(* PLC project Untitled6.project, CODESYS CODESYS V3.5 SP20 *)
(* stored: creationDateTime 2025-11-22T16:58:05.889821, modificationDateTime 2025-11-22T16:57:51.3762535 *)

TYPE ST_MotionState : STRUCT
  fDuration : LREAL := 0.0;  (* Duration of this segment *)
  fPos : LREAL := 0.0;  (* Position *)
  fVel : LREAL := 0.0;  (* Velocity *)
  fAcc : LREAL := 0.0;  (* Acceleration *)
  fJerk : LREAL := 0.0;  (* Jerk *)
END_STRUCT;
END_TYPE

TYPE ST_MotionLimits : STRUCT
  fVelMax : LREAL;
  fAccMax : LREAL;
  fJerkMax : LREAL;
END_STRUCT;
END_TYPE

FUNCTION FC_S7RTT_CalcTrajDist : LREAL
  VAR_INPUT
    v_peak : LREAL;
    start_v : LREAL;
    start_a : LREAL;
    target_v : LREAL;
    a_max : LREAL;
    j_max : LREAL;
  END_VAR
  VAR
    t_buf : ARRAY[1..5] OF LREAL;
    j_buf : ARRAY[1..5] OF LREAL;
    cnt : INT;
    i : INT;
    v_curr : LREAL;
    a_curr : LREAL;
    dist_total : LREAL;
    t_seg : LREAL;
    j_seg : LREAL;
  END_VAR

            dist_total := 0.0;
v_curr := start_v;
a_curr := start_a;

// Phase 1: Start -> Peak Velocity
cnt := FC_S7RTT_BuildProfile(v_curr, a_curr, v_peak, a_max, j_max, t_buf, j_buf);
FOR i := 1 TO cnt DO
	t_seg := t_buf[i];
	j_seg := j_buf[i];
    // Standard kinematic integration: p = p0 + v0*t + 0.5*a0*t^2 + 1/6*j*t^3
	dist_total := dist_total + v_curr * t_seg + 0.5 * a_curr * t_seg*t_seg + (1.0/6.0) * j_seg * t_seg*t_seg*t_seg;
	v_curr := v_curr + a_curr * t_seg + 0.5 * j_seg * t_seg*t_seg;
	a_curr := a_curr + j_seg * t_seg;
END_FOR;

// Phase 2: Peak Velocity -> Target Velocity
cnt := FC_S7RTT_BuildProfile(v_curr, a_curr, target_v, a_max, j_max, t_buf, j_buf);
FOR i := 1 TO cnt DO
	t_seg := t_buf[i];
	j_seg := j_buf[i];
	dist_total := dist_total + v_curr * t_seg + 0.5 * a_curr * t_seg*t_seg + (1.0/6.0) * j_seg * t_seg*t_seg*t_seg;
	v_curr := v_curr + a_curr * t_seg + 0.5 * j_seg * t_seg*t_seg;
	a_curr := a_curr + j_seg * t_seg;
END_FOR;

FC_S7RTT_CalcTrajDist := dist_total;
          
END_FUNCTION

FUNCTION_BLOCK FB_S7RTT_Plan
  VAR_INPUT
    Execute : BOOL;
    ModeVelocity : BOOL;
    StartState : ST_MotionState;
    TargetPos : LREAL;
    TargetVel : LREAL;
    Limits : ST_MotionLimits;
  END_VAR
  VAR_OUTPUT
    Done : BOOL;
    Error : BOOL;
    SegmentCount : INT;
    Trajectory : ARRAY[1..32] OF ST_MotionState;
  END_VAR
  VAR
    trig_exec : BOOL;
    prev_exec : BOOL;
    c_pos : LREAL;
    c_vel : LREAL;
    c_acc : LREAL;
    dist_req : LREAL;
    iter : INT;
    sa : LREAL;
    sb : LREAL;
    sc : LREAL;
    fa : LREAL;
    fb : LREAL;
    fc : LREAL;
    sd : LREAL;
    se : LREAL;
    tol1 : LREAL;
    xm : LREAL;
    fCoefP : LREAL;
    fCoefQ : LREAL;
    fCoefR : LREAL;
    fCoefS : LREAL;
    min1 : LREAL;
    min2 : LREAL;
    mflag : BOOL;
    best_v : LREAL;
    t_shape_buf : ARRAY[1..5] OF LREAL;
    j_shape_buf : ARRAY[1..5] OF LREAL;
    shape_cnt : INT;
    i : INT;
    t_rec : LREAL;
    d_upper : LREAL;
    d_lower : LREAL;
    d_inertial : LREAL;
    v_inertial : LREAL;
    j_restore : LREAL;
    t_to_zero : LREAL;
    gap : LREAL;
    t_cruise : LREAL;
    v_mid : LREAL;
    a_mid : LREAL;
    EPS_TIME : LREAL := 1E-09;
    EPS_VAL : LREAL := 1E-07;
    EPS_ACC : LREAL := 1E-06;
    EPS_DIST : LREAL := 1E-08;
    SOLVER_TOL : LREAL := 1E-08;
    SOLVER_EPS : LREAL := 2.22E-16;
    MAX_ITER : INT := 100;
    ref_idx : INT;
    max_dt : LREAL;
    dt_fix : LREAL;
    v_cruise_start : LREAL;
    new_dt : LREAL;
  END_VAR

            // ==============================================================================
// File Name:    FB_S7RTT_Plan.st
// Author:       feecat
// Version:      V1.6.1
// Description:  Simple 7seg Real-Time Trajectory Generator
// Website:      https://github.com/feecat/S7RTT
// License:      Apache License Version 2.0
// ==============================================================================
//
// Licensed under the Apache License, Version 2.0 (the "License");
// you may not use this file except in compliance with the License.
// You may obtain a copy of the License at
//
//     http://www.apache.org/licenses/LICENSE-2.0
//
// Unless required by applicable law or agreed to in writing, software
// distributed under the License is distributed on an "AS IS" BASIS,
// WITHOUT WARRANTIES OR CONDITIONS OF ANY KIND, either express or implied.
// See the License for the specific language governing permissions and
// limitations under the License.
// ==============================================================================

trig_exec := Execute AND NOT prev_exec;
prev_exec := Execute;

IF NOT Execute THEN
	Done := FALSE;
	Error := FALSE;
	RETURN;
END_IF

IF NOT trig_exec THEN
	RETURN;
END_IF;

// --- Initialization ---
Done := FALSE;
Error := FALSE;
SegmentCount := 0;

IF Limits.fVelMax <= 0.0 OR Limits.fAccMax <= 0.0 OR Limits.fJerkMax <= 0.0 THEN
	Error := TRUE;
	RETURN;
END_IF;

c_pos := StartState.fPos;
c_vel := StartState.fVel;
c_acc := StartState.fAcc;

// ========================================================
// 1. Acceleration Recovery (Safety Decel to Max Limits)
// ========================================================
IF c_acc > Limits.fAccMax + EPS_VAL THEN
	t_rec := (c_acc - Limits.fAccMax) / Limits.fJerkMax;
	SegmentCount := SegmentCount + 1;
	Trajectory[SegmentCount].fDuration := t_rec;
	Trajectory[SegmentCount].fJerk     := -Limits.fJerkMax;
	
	// Integrate state forward
	c_pos := c_pos + c_vel * t_rec + 0.5 * c_acc * t_rec*t_rec + (1.0/6.0) * (-Limits.fJerkMax) * t_rec*t_rec*t_rec;
	c_vel := c_vel + c_acc * t_rec + 0.5 * (-Limits.fJerkMax) * t_rec*t_rec;
	c_acc := Limits.fAccMax;
	
ELSIF c_acc < -Limits.fAccMax - EPS_VAL THEN
	t_rec := (-Limits.fAccMax - c_acc) / Limits.fJerkMax;
	SegmentCount := SegmentCount + 1;
	Trajectory[SegmentCount].fDuration := t_rec;
	Trajectory[SegmentCount].fJerk     := Limits.fJerkMax;
	
	// Integrate state forward
	c_pos := c_pos + c_vel * t_rec + 0.5 * c_acc * t_rec*t_rec + (1.0/6.0) * (Limits.fJerkMax) * t_rec*t_rec*t_rec;
	c_vel := c_vel + c_acc * t_rec + 0.5 * (Limits.fJerkMax) * t_rec*t_rec;
	c_acc := -Limits.fAccMax;
END_IF;

// ========================================================
// 2. Plan Generation
// ========================================================

IF ModeVelocity THEN
	// ---------------- Velocity Mode ----------------
	v_mid := TargetVel; 
	IF v_mid > Limits.fVelMax THEN v_mid := Limits.fVelMax; END_IF;
	IF v_mid < -Limits.fVelMax THEN v_mid := -Limits.fVelMax; END_IF;

	shape_cnt := FC_S7RTT_BuildProfile(c_vel, c_acc, v_mid, Limits.fAccMax, Limits.fJerkMax, t_shape_buf, j_shape_buf);
	
	FOR i := 1 TO shape_cnt DO
		IF SegmentCount < 32 THEN
			SegmentCount := SegmentCount + 1;
			Trajectory[SegmentCount].fDuration := t_shape_buf[i];
			Trajectory[SegmentCount].fJerk     := j_shape_buf[i];
		END_IF;
	END_FOR;

ELSE
	// ---------------- Position Mode ----------------
	dist_req := TargetPos - c_pos;
	
	// Calculate Inertial Velocity (Peak velocity if we stopped now)
	t_to_zero := ABS(c_acc) / Limits.fJerkMax;
	IF c_acc > 0.0 THEN j_restore := -Limits.fJerkMax; ELSE j_restore := Limits.fJerkMax; END_IF;
	v_inertial := c_vel + c_acc * t_to_zero + 0.5 * j_restore * t_to_zero * t_to_zero;

	// Check 1: Max Reach Checks (Can we physically reach the target?)
	// This determines if we need to cruise at VMax
	d_upper := FC_S7RTT_CalcTrajDist(Limits.fVelMax, c_vel, c_acc, TargetVel, Limits.fAccMax, Limits.fJerkMax);
	d_lower := FC_S7RTT_CalcTrajDist(-Limits.fVelMax, c_vel, c_acc, TargetVel, Limits.fAccMax, Limits.fJerkMax);

	IF dist_req > d_upper + EPS_DIST THEN
		// Case: Cruise Positive (Go to Vmax, Cruise, then Decel)
		gap := dist_req - d_upper;
		t_cruise := gap / Limits.fVelMax;
		
		// 1. Start -> Vmax
		shape_cnt := FC_S7RTT_BuildProfile(c_vel, c_acc, Limits.fVelMax, Limits.fAccMax, Limits.fJerkMax, t_shape_buf, j_shape_buf);
		
		// Add Cruise Segment
		IF t_cruise > EPS_TIME THEN
		   shape_cnt := shape_cnt + 1;
		   t_shape_buf[shape_cnt] := t_cruise;
		   j_shape_buf[shape_cnt] := 0.0;
		END_IF;
		
		// Integ & Append
		v_mid := c_vel; a_mid := c_acc;
		FOR i := 1 TO shape_cnt DO
			IF SegmentCount < 32 THEN
				SegmentCount := SegmentCount + 1;
				Trajectory[SegmentCount].fDuration := t_shape_buf[i];
				Trajectory[SegmentCount].fJerk     := j_shape_buf[i];
				v_mid := v_mid + a_mid * t_shape_buf[i] + 0.5 * j_shape_buf[i] * t_shape_buf[i]*t_shape_buf[i];
				a_mid := a_mid + j_shape_buf[i] * t_shape_buf[i];
			END_IF;
		END_FOR;
		
		// 2. Vmax -> Target
		shape_cnt := FC_S7RTT_BuildProfile(v_mid, a_mid, TargetVel, Limits.fAccMax, Limits.fJerkMax, t_shape_buf, j_shape_buf);
		FOR i := 1 TO shape_cnt DO
			IF SegmentCount < 32 THEN
				SegmentCount := SegmentCount + 1;
				Trajectory[SegmentCount].fDuration := t_shape_buf[i];
				Trajectory[SegmentCount].fJerk     := j_shape_buf[i];
			END_IF;
		END_FOR;

	ELSIF dist_req < d_lower - EPS_DIST THEN
		// Case: Cruise Negative
		gap := dist_req - d_lower;
		t_cruise := gap / (-Limits.fVelMax);
		
		// 1. Start -> -Vmax
		shape_cnt := FC_S7RTT_BuildProfile(c_vel, c_acc, -Limits.fVelMax, Limits.fAccMax, Limits.fJerkMax, t_shape_buf, j_shape_buf);
		
		IF t_cruise > EPS_TIME THEN
		   shape_cnt := shape_cnt + 1;
		   t_shape_buf[shape_cnt] := t_cruise;
		   j_shape_buf[shape_cnt] := 0.0;
		END_IF;
		
		v_mid := c_vel; a_mid := c_acc;
		FOR i := 1 TO shape_cnt DO
			IF SegmentCount < 32 THEN
				SegmentCount := SegmentCount + 1;
				Trajectory[SegmentCount].fDuration := t_shape_buf[i];
				Trajectory[SegmentCount].fJerk     := j_shape_buf[i];
				v_mid := v_mid + a_mid * t_shape_buf[i] + 0.5 * j_shape_buf[i] * t_shape_buf[i]*t_shape_buf[i];
				a_mid := a_mid + j_shape_buf[i] * t_shape_buf[i];
			END_IF;
		END_FOR;
		
		// 2. -Vmax -> Target
		shape_cnt := FC_S7RTT_BuildProfile(v_mid, a_mid, TargetVel, Limits.fAccMax, Limits.fJerkMax, t_shape_buf, j_shape_buf);
		FOR i := 1 TO shape_cnt DO
			IF SegmentCount < 32 THEN
				SegmentCount := SegmentCount + 1;
				Trajectory[SegmentCount].fDuration := t_shape_buf[i];
				Trajectory[SegmentCount].fJerk     := j_shape_buf[i];
			END_IF;
		END_FOR;

	ELSE
		// Case: Target is reachable without cruising at limits. 
		// We need to find the peak velocity 'v_peak' that produces the exact distance.
		
		d_inertial := FC_S7RTT_CalcTrajDist(v_inertial, c_vel, c_acc, TargetVel, Limits.fAccMax, Limits.fJerkMax);
		
		// Define search brackets for Brent's method [sa, sb]
		// Logic: If requested distance > inertial distance, we need to go faster/more positive.
		IF dist_req > d_inertial THEN
			sa := v_inertial - (10.0 * EPS_VAL);
			sb := MAX(Limits.fVelMax, MAX(ABS(c_vel), ABS(TargetVel))) * 1.5 + 10.0;
		ELSE
			sb := v_inertial + (10.0 * EPS_VAL);
			sa := -(MAX(Limits.fVelMax, MAX(ABS(c_vel), ABS(TargetVel))) * 1.5 + 10.0);
		END_IF;
		
		IF sa >= sb THEN sa := sb - EPS_VAL; END_IF;
		
		// Function evaluation at endpoints
		fa := FC_S7RTT_CalcTrajDist(sa, c_vel, c_acc, TargetVel, Limits.fAccMax, Limits.fJerkMax) - dist_req;
		fb := FC_S7RTT_CalcTrajDist(sb, c_vel, c_acc, TargetVel, Limits.fAccMax, Limits.fJerkMax) - dist_req;
		
		IF (fa > 0.0 AND fb > 0.0) OR (fa < 0.0 AND fb < 0.0) THEN
			// Error: Root not bracketed. Use the best guess.
			IF ABS(fa) < ABS(fb) THEN best_v := sa; ELSE best_v := sb; END_IF;
		ELSE
			// Brent's Method Solver
			sc := sa; fc := fa; sd := sb - sa; se := sd; mflag := TRUE;
			
			FOR iter := 1 TO MAX_ITER DO
				 IF ABS(fc) < ABS(fb) THEN
					sa := sb; sb := sc; sc := sa;
					fa := fb; fb := fc; fc := fa;
				 END_IF;
				 
				 tol1 := 2.0 * SOLVER_EPS * ABS(sb) + 0.5 * SOLVER_TOL;
				 xm := 0.5 * (sc - sb);
				 
				 IF ABS(xm) <= tol1 OR ABS(fb) < SOLVER_TOL THEN
					EXIT; // Converged
				 END_IF;
				 
				 IF ABS(se) >= tol1 AND ABS(fa) > ABS(fb) THEN
					fCoefS := fb / fa;
					IF sa = sc THEN
						fCoefP := 2.0 * xm * fCoefS;
						fCoefQ := 1.0 - fCoefS;
					ELSE
						fCoefQ := fa / fc; fCoefR := fb / fc;
						fCoefP := fCoefS * (2.0 * xm * fCoefQ * (fCoefQ - fCoefR) - (sb - sa) * (fCoefR - 1.0));
						fCoefQ := (fCoefQ - 1.0) * (fCoefR - 1.0) * (fCoefS - 1.0);
					END_IF;
					
					IF fCoefP > 0.0 THEN fCoefQ := -fCoefQ; END_IF;
					fCoefP := ABS(fCoefP);
					min1 := 3.0 * xm * fCoefQ - ABS(tol1 * fCoefQ);
					min2 := ABS(se * fCoefQ);
					
					IF 2.0 * fCoefP < min1 THEN
						IF mflag THEN
							IF 2.0 * fCoefP < min2 THEN se := sd; sd := fCoefP / fCoefQ; mflag := FALSE;
							ELSE sd := xm; se := sd; mflag := TRUE; END_IF;
						ELSE
							IF 2.0 * fCoefP < ABS(sd * fCoefQ) THEN se := sd; sd := fCoefP / fCoefQ; mflag := FALSE;
							ELSE sd := xm; se := sd; mflag := TRUE; END_IF;
						END_IF;
					ELSE
						sd := xm; se := sd; mflag := TRUE;
					END_IF;
				 ELSE
					 sd := xm; se := sd; mflag := TRUE;
				 END_IF;
				 
				 sa := sb; fa := fb;
				 
				 IF ABS(sd) > tol1 THEN
					sb := sb + sd;
				 ELSE
					IF xm > 0.0 THEN sb := sb + tol1; ELSE sb := sb - tol1; END_IF;
				 END_IF;
				 
				 fb := FC_S7RTT_CalcTrajDist(sb, c_vel, c_acc, TargetVel, Limits.fAccMax, Limits.fJerkMax) - dist_req;
				 
				 IF (fb > 0.0 AND fc > 0.0) OR (fb < 0.0 AND fc < 0.0) THEN
					 sc := sa; fc := fa; sd := sb - sa; se := sd; mflag := TRUE;
				 END_IF;
			END_FOR;
			best_v := sb;
		END_IF;
		
		// Generate final trajectory using the solved velocity
		// 1. Start -> v_peak
		shape_cnt := FC_S7RTT_BuildProfile(c_vel, c_acc, best_v, Limits.fAccMax, Limits.fJerkMax, t_shape_buf, j_shape_buf);
		v_mid := c_vel; a_mid := c_acc;
		FOR i := 1 TO shape_cnt DO
			IF SegmentCount < 32 THEN
				SegmentCount := SegmentCount + 1;
				Trajectory[SegmentCount].fDuration := t_shape_buf[i];
				Trajectory[SegmentCount].fJerk     := j_shape_buf[i];
				v_mid := v_mid + a_mid * t_shape_buf[i] + 0.5 * j_shape_buf[i] * t_shape_buf[i]*t_shape_buf[i];
				a_mid := a_mid + j_shape_buf[i] * t_shape_buf[i];
			END_IF;
		END_FOR;
		
		// 2. v_peak -> Target
		shape_cnt := FC_S7RTT_BuildProfile(v_mid, a_mid, TargetVel, Limits.fAccMax, Limits.fJerkMax, t_shape_buf, j_shape_buf);
		FOR i := 1 TO shape_cnt DO
			IF SegmentCount < 32 THEN
				SegmentCount := SegmentCount + 1;
				Trajectory[SegmentCount].fDuration := t_shape_buf[i];
				Trajectory[SegmentCount].fJerk     := j_shape_buf[i];
			END_IF;
		END_FOR;
	END_IF; // End Bounds Checks
END_IF; // End ModeVelocity
// ========================================================
// 2.5. Trajectory Refinement (Fix Integration Drift)
// ========================================================
// Only perform refinement if we have segments and are in Position Mode
IF SegmentCount > 0 AND NOT ModeVelocity THEN
	c_pos := StartState.fPos;
	c_vel := StartState.fVel;
	c_acc := StartState.fAcc;
	
	// Variables for refinement search
	// You need to declare: 
	// ref_idx: INT; max_dt: LREAL; sim_p: LREAL; 
	// dt_fix: LREAL; v_cruise_start: LREAL;
	
	ref_idx := -1;
	max_dt := -1.0;
	
	FOR i := 1 TO SegmentCount DO
		t_rec := Trajectory[i].fDuration;
		j_restore := Trajectory[i].fJerk;
		
		// Check for Constant Velocity segment (J=0, A approx 0)
		// We simulate A at the START of the segment
		IF ABS(j_restore) < SOLVER_EPS AND ABS(c_acc) < EPS_ACC THEN
			IF t_rec > max_dt THEN
				max_dt := t_rec;
				ref_idx := i;
				v_cruise_start := c_vel; // Store velocity of this segment
			END_IF;
		END_IF;
		
		// Integrate to next state
		c_pos := c_pos + c_vel * t_rec + 0.5 * c_acc * t_rec*t_rec + (1.0/6.0) * j_restore * t_rec*t_rec*t_rec;
		c_vel := c_vel + c_acc * t_rec + 0.5 * j_restore * t_rec*t_rec;
		c_acc := c_acc + j_restore * t_rec;
	END_FOR;
	
	// Calculate Error based on simulated final position
	gap := TargetPos - c_pos;
	
	// Apply fix if we found a suitable cruise segment and error exists
	IF ref_idx <> -1 AND ABS(gap) > EPS_DIST AND ABS(v_cruise_start) > EPS_VAL THEN
		dt_fix := gap / v_cruise_start;
		Trajectory[ref_idx].fDuration := Trajectory[ref_idx].fDuration + dt_fix;
		
		// Safety: prevent negative time
		IF Trajectory[ref_idx].fDuration < EPS_TIME THEN 
			Trajectory[ref_idx].fDuration := EPS_TIME; 
		END_IF;
	END_IF;
END_IF;

// ========================================================
// 3. Final Pass: Calculate Absolute Positions
// ========================================================
c_pos := StartState.fPos; 
c_vel := StartState.fVel; 
c_acc := StartState.fAcc;

FOR i := 1 TO SegmentCount DO
	// Store the starting state of this segment
	Trajectory[i].fPos := c_pos;
	Trajectory[i].fVel := c_vel;
	Trajectory[i].fAcc := c_acc;
	
	t_rec := Trajectory[i].fDuration;
	j_restore := Trajectory[i].fJerk;
	
	c_pos := c_pos + c_vel * t_rec + 0.5 * c_acc * t_rec*t_rec + (1.0/6.0) * j_restore * t_rec*t_rec*t_rec;
	c_vel := c_vel + c_acc * t_rec + 0.5 * j_restore * t_rec*t_rec;
	c_acc := c_acc + j_restore * t_rec;
END_FOR;

Done := TRUE;
          
END_FUNCTION_BLOCK

FUNCTION FC_S7RTT_AtTime : ST_MotionState
  VAR_INPUT
    Trajectory : ARRAY[1..32] OF ST_MotionState;
    SegCount : INT;
    ElapsedTime : LREAL;
  END_VAR
  VAR
    i : INT;
    t_rem : LREAL;
    t : LREAL;
    j : LREAL;
    p0 : LREAL;
    v0 : LREAL;
    a0 : LREAL;
    last_idx : INT;
  END_VAR

            IF SegCount <= 0 THEN
    // No trajectory, return zero/empty state
    FC_S7RTT_AtTime.fPos := 0.0; FC_S7RTT_AtTime.fVel := 0.0; FC_S7RTT_AtTime.fAcc := 0.0;
    RETURN;
END_IF;

IF ElapsedTime <= 0.0 THEN
     // Return Initial State from First Segment
     FC_S7RTT_AtTime := Trajectory[1]; 
     FC_S7RTT_AtTime.fDuration := 0.0;
     FC_S7RTT_AtTime.fJerk := 0.0;
     RETURN;
END_IF;

t_rem := ElapsedTime;

FOR i := 1 TO SegCount DO
	IF t_rem <= Trajectory[i].fDuration THEN
		t := t_rem;
		j := Trajectory[i].fJerk;
		// Use pre-calculated state at segment start
		p0 := Trajectory[i].fPos;
		v0 := Trajectory[i].fVel;
		a0 := Trajectory[i].fAcc;

		FC_S7RTT_AtTime.fPos := p0 + v0 * t + 0.5 * a0 * t*t + (1.0/6.0) * j * t*t*t;
		FC_S7RTT_AtTime.fVel := v0 + a0 * t + 0.5 * j * t*t;
		FC_S7RTT_AtTime.fAcc := a0 + j * t;
		FC_S7RTT_AtTime.fJerk := j;
		FC_S7RTT_AtTime.fDuration := 0.0;
		RETURN;
	ELSE
		t_rem := t_rem - Trajectory[i].fDuration;
	END_IF;
END_FOR;

// Time is beyond end of trajectory
// Calculate Final State of last segment
last_idx := SegCount;
t := Trajectory[last_idx].fDuration;
j := Trajectory[last_idx].fJerk;
p0 := Trajectory[last_idx].fPos;
v0 := Trajectory[last_idx].fVel;
a0 := Trajectory[last_idx].fAcc;

p0 := p0 + v0 * t + 0.5 * a0 * t*t + (1.0/6.0) * j * t*t*t;
v0 := v0 + a0 * t + 0.5 * j * t*t;

// Hold Final Position (assuming v=target, a=0 at end)
// Linear projection if Velocity is non-zero
FC_S7RTT_AtTime.fPos := p0 + v0 * t_rem;
FC_S7RTT_AtTime.fVel := v0;
FC_S7RTT_AtTime.fAcc := 0.0;
FC_S7RTT_AtTime.fJerk := 0.0;
FC_S7RTT_AtTime.fDuration := 0.0;
          
END_FUNCTION

FUNCTION FC_S7RTT_BuildProfile : INT
  VAR_INPUT
    in_v_start : LREAL;
    in_a_start : LREAL;
    in_v_target : LREAL;
    in_a_max : LREAL;
    in_j_max : LREAL;
  END_VAR
  VAR_IN_OUT
    out_time : ARRAY[1..5] OF LREAL;
    out_jerk : ARRAY[1..5] OF LREAL;
  END_VAR
  VAR
    acc_clamped : LREAL;
    t_to_zero : LREAL;
    j_restore : LREAL;
    v_min_feasible : LREAL;
    direction : LREAL;
    v0_mod : LREAL;
    a0_mod : LREAL;
    v1_mod : LREAL;
    t1_max : LREAL;
    t3_max : LREAL;
    dv_inflection : LREAL;
    dv_req : LREAL;
    dv_missing : LREAL;
    term : LREAL;
    a_peak : LREAL;
    t1 : LREAL;
    t2 : LREAL;
    t3 : LREAL;
    cnt : INT;
    EPS : LREAL := 1E-09;
  END_VAR

            cnt := 0;

// 1. Clamp initial acceleration to limits
acc_clamped := in_a_start;
IF acc_clamped > in_a_max THEN acc_clamped := in_a_max; END_IF;
IF acc_clamped < -in_a_max THEN acc_clamped := -in_a_max; END_IF;

// 2. Check feasibility (can we stop?)
t_to_zero := ABS(acc_clamped) / in_j_max;
IF ABS(acc_clamped) > EPS THEN
    IF acc_clamped > 0.0 THEN j_restore := -in_j_max; ELSE j_restore := in_j_max; END_IF;
ELSE
    j_restore := 0.0;
END_IF;

v_min_feasible := in_v_start + acc_clamped * t_to_zero + 0.5 * j_restore * t_to_zero * t_to_zero;

// 3. Determine direction
direction := 1.0;
IF in_v_target < v_min_feasible - EPS THEN
    direction := -1.0;
END_IF;

// 4. Normalize to positive quadrant
v0_mod := in_v_start * direction;
a0_mod := acc_clamped * direction;
v1_mod := in_v_target * direction;

t1_max := (in_a_max - a0_mod) / in_j_max;
IF t1_max < 0.0 THEN t1_max := 0.0; END_IF;

t3_max := in_a_max / in_j_max;

// Velocity change at inflection (max accel reached)
dv_inflection := (a0_mod * t1_max + 0.5 * in_j_max * t1_max * t1_max) +
                 (in_a_max * t3_max - 0.5 * in_j_max * t3_max * t3_max);

dv_req := v1_mod - v0_mod;

// 5. Calculate profile times
IF dv_req > dv_inflection THEN
    // Trapezoidal (Constant Acceleration Phase)
    dv_missing := dv_req - dv_inflection;
    t2 := dv_missing / in_a_max;
    t1 := t1_max;
    t3 := t3_max;
ELSE
    // Triangular (No Constant Acceleration)
    term := in_j_max * dv_req + 0.5 * a0_mod * a0_mod;
    IF term < 0.0 THEN term := 0.0; END_IF;
    a_peak := SQRT(term);
    
    t1 := (a_peak - a0_mod) / in_j_max;
    IF t1 < 0.0 THEN t1 := 0.0; END_IF;
    
    t3 := a_peak / in_j_max;
    IF t3 < 0.0 THEN t3 := 0.0; END_IF;
    
    t2 := 0.0;
END_IF;

// 6. Output Segments
IF t1 > EPS THEN
    cnt := cnt + 1; out_time[cnt] := t1; out_jerk[cnt] := direction * in_j_max;
END_IF;
IF t2 > EPS THEN
    cnt := cnt + 1; out_time[cnt] := t2; out_jerk[cnt] := 0.0;
END_IF;
IF t3 > EPS THEN
    cnt := cnt + 1; out_time[cnt] := t3; out_jerk[cnt] := -direction * in_j_max;
END_IF;

FC_S7RTT_BuildProfile := cnt;
          
END_FUNCTION

FUNCTION_BLOCK FB_S7RTT_Plan_Velocity
  VAR_INPUT
    Execute : BOOL;
    StartState : ST_MotionState;
    TargetVel : LREAL;
    Limits : ST_MotionLimits;
  END_VAR
  VAR_OUTPUT
    Done : BOOL;
    Error : BOOL;
    SegmentCount : INT;
    Trajectory : ARRAY[1..32] OF ST_MotionState;
  END_VAR
  VAR
    trig_exec : BOOL;
    prev_exec : BOOL;
    c_pos : LREAL;
    c_vel : LREAL;
    c_acc : LREAL;
    t_rec : LREAL;
    safe_target_v : LREAL;
    t_shape_buf : ARRAY[1..5] OF LREAL;
    j_shape_buf : ARRAY[1..5] OF LREAL;
    shape_cnt : INT;
    i : INT;
    j_restore : LREAL;
    EPS_VAL : LREAL := 1E-07;
  END_VAR

            trig_exec := Execute AND NOT prev_exec;
prev_exec := Execute;

IF NOT Execute THEN
	Done := FALSE;
	Error := FALSE;
	RETURN;
END_IF

IF NOT trig_exec THEN
    RETURN;
END_IF;

// --- Initialization ---
Done := FALSE;
Error := FALSE;
SegmentCount := 0;

IF Limits.fVelMax <= 0.0 OR Limits.fAccMax <= 0.0 OR Limits.fJerkMax <= 0.0 THEN
    Error := TRUE;
    RETURN;
END_IF;

// Load internal state
c_pos := StartState.fPos;
c_vel := StartState.fVel;
c_acc := StartState.fAcc;

// ========================================================
// 1. Safety Deceleration (Handle Initial Accel Overload)
// ========================================================
IF c_acc > Limits.fAccMax + EPS_VAL THEN
    // Case: Accel too high positive, pull down with negative jerk
    t_rec := (c_acc - Limits.fAccMax) / Limits.fJerkMax;
    IF t_rec > 0.0 THEN
        SegmentCount := SegmentCount + 1;
        Trajectory[SegmentCount].fDuration := t_rec;
        Trajectory[SegmentCount].fJerk     := -Limits.fJerkMax;
        
        // Integrate state forward
        c_pos := c_pos + c_vel * t_rec + 0.5 * c_acc * t_rec*t_rec + (1.0/6.0) * (-Limits.fJerkMax) * t_rec*t_rec*t_rec;
        c_vel := c_vel + c_acc * t_rec + 0.5 * (-Limits.fJerkMax) * t_rec*t_rec;
        c_acc := Limits.fAccMax; // Clamp to avoid drift
    END_IF;
    
ELSIF c_acc < -Limits.fAccMax - EPS_VAL THEN
    // Case: Accel too high negative, pull up with positive jerk
    t_rec := (-Limits.fAccMax - c_acc) / Limits.fJerkMax;
    IF t_rec > 0.0 THEN
        SegmentCount := SegmentCount + 1;
        Trajectory[SegmentCount].fDuration := t_rec;
        Trajectory[SegmentCount].fJerk     := Limits.fJerkMax;
        
        // Integrate state forward
        c_pos := c_pos + c_vel * t_rec + 0.5 * c_acc * t_rec*t_rec + (1.0/6.0) * (Limits.fJerkMax) * t_rec*t_rec*t_rec;
        c_vel := c_vel + c_acc * t_rec + 0.5 * (Limits.fJerkMax) * t_rec*t_rec;
        c_acc := -Limits.fAccMax; // Clamp
    END_IF;
END_IF;

// ========================================================
// 2. Clamp Target Velocity
// ========================================================
safe_target_v := TargetVel;
IF safe_target_v > Limits.fVelMax THEN safe_target_v := Limits.fVelMax; END_IF;
IF safe_target_v < -Limits.fVelMax THEN safe_target_v := -Limits.fVelMax; END_IF;

// ========================================================
// 3. Build Velocity Profile
// ========================================================
// Uses the helper function to calculate S-Curve times
shape_cnt := FC_S7RTT_BuildProfile(c_vel, c_acc, safe_target_v, Limits.fAccMax, Limits.fJerkMax, t_shape_buf, j_shape_buf);

FOR i := 1 TO shape_cnt DO
    IF SegmentCount < 32 THEN
        SegmentCount := SegmentCount + 1;
        Trajectory[SegmentCount].fDuration := t_shape_buf[i];
        Trajectory[SegmentCount].fJerk     := j_shape_buf[i];
    END_IF;
END_FOR;

// ========================================================
// 4. Final Pass: Calculate Absolute Positions for Nodes
// ========================================================
// Re-run integration from start to fill in P/V/A for output array
c_pos := StartState.fPos; 
c_vel := StartState.fVel; 
c_acc := StartState.fAcc;

FOR i := 1 TO SegmentCount DO
    // Store the starting state of this segment into the array
    Trajectory[i].fPos := c_pos;
    Trajectory[i].fVel := c_vel;
    Trajectory[i].fAcc := c_acc;
    
    t_rec := Trajectory[i].fDuration;
    j_restore := Trajectory[i].fJerk;
    
    // Integrate to find start state for NEXT segment
    c_pos := c_pos + c_vel * t_rec + 0.5 * c_acc * t_rec*t_rec + (1.0/6.0) * j_restore * t_rec*t_rec*t_rec;
    c_vel := c_vel + c_acc * t_rec + 0.5 * j_restore * t_rec*t_rec;
    c_acc := c_acc + j_restore * t_rec;
END_FOR;

Done := TRUE;
          
END_FUNCTION_BLOCK
